// TIA Portal project "E01_KOP_SCL" (V18)

(* hardware
DEVICE "S71500/ET200MP station_1"  S7-1500 station
   slot 0: "Telaio di montaggio_0"  Rack  6ES7 590-1***0-0AA0
   slot 1: "PLC_1"  CPU 1516-3 PN/DP  6ES7 516-3AN01-0AB0  V2.5
      slot 3: "Display CPU_1"  6ES7591-1BA00-0AA0
   slot 2: "DI 32x24VDC HF_1"  DI 32x24VDC HF  6ES7 521-1BL00-0AB0  V2.1
   slot 3: "DQ 32x24VDC/0.5A HF_1"  DQ 32x24VDC/0.5A HF  6ES7 522-1BL01-0AB0  V1.0
   slot 4: "AI 8xU/I/RTD/TC ST_1"  AI 8xU/I/RTD/TC ST  6ES7 531-7KF00-0AB0  V2.1
   slot 5: "AQ 4xU/I ST_1"  AQ 4xU/I ST  6ES7 532-5HD00-0AB0  V2.1
*)

// ===== PLC "PLC_1"  CPU 1516-3 PN/DP =====

VAR_GLOBAL   // PLC tag table "Tabella delle variabili standard"
   "Led 1" AT %Q3.0 : Bool;
   "Led 2" AT %Q3.1 : Bool;
   "Led 3" AT %Q3.2 : Bool;
   "Led 4" AT %Q3.3 : Bool;
   "Led 5" AT %Q3.4 : Bool;
   "Led 6" AT %Q3.5 : Bool;
   "Led 7" AT %Q3.6 : Bool;
   "Led 8" AT %Q3.7 : Bool;
END_VAR

DATA_BLOCK "DB_dati"   // DB1
{ S7_Optimized_Access := 'TRUE' }
VERSION : 0.1
   VAR
      btn1 : Bool;
      btn2 : Bool;
      btn3 : Bool;
      btn4 : Bool;
      btn5 : Bool;
      btn6 : Bool;
      btn7 : Bool;
      btn8 : Bool;
   END_VAR
BEGIN
END_DATA_BLOCK

FUNCTION "FC_KOP" : Void   // FC1, LAD
{ S7_Optimized_Access := 'TRUE' }
VERSION : 0.1
BEGIN

REGION Network 1
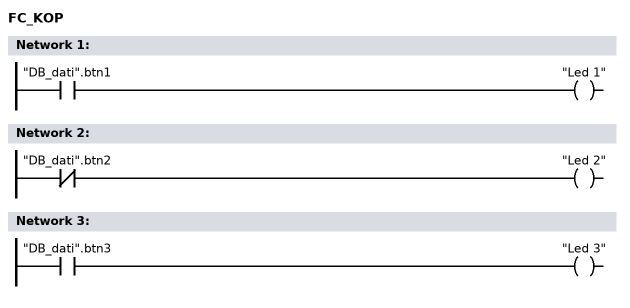
   RUNG wire#powerrail
      Contact( "DB_dati".btn1 )
      Coil( "Led 1" )
   END_RUNG
   // the same network as SCL:
   "Led 1" := "DB_dati".btn1;
END_REGION

REGION Network 2
   RUNG wire#powerrail
      I_Contact( "DB_dati".btn2 )
      Coil( "Led 2" )
   END_RUNG
   // the same network as SCL:
   "Led 2" := NOT "DB_dati".btn2;
END_REGION

REGION Network 3
   RUNG wire#powerrail
      Contact( "DB_dati".btn3 )
      Coil( "Led 3" )
   END_RUNG
   // the same network as SCL:
   "Led 3" := "DB_dati".btn3;
END_REGION
END_FUNCTION

FUNCTION "FC_SCL" : Void   // FC2, SCL
{ S7_Optimized_Access := 'TRUE' }
VERSION : 0.1
BEGIN
   IF "DB_dati".btn4 = TRUE THEN
       "Led 4" := TRUE;
   ELSE
       "Led 4" := FALSE;
   END_IF;
   //Commenti 
   IF "DB_dati".btn5 = FALSE THEN
       "Led 5" := TRUE;
   ELSE
       "Led 5" := FALSE;
   END_IF;
   //
   IF "DB_dati".btn6 = TRUE THEN
       "Led 6" := TRUE;
   ELSE
       "Led 6" := FALSE;
   END_IF;
END_FUNCTION

ORGANIZATION_BLOCK "Main"   // OB1, LAD, ProgramCycle
TITLE = "Main Program Sweep (Cycle)"
{ S7_Optimized_Access := 'TRUE' }
VERSION : 0.1
   VAR_INPUT
      Initial_Call : Bool;   // Initial call of this OB
      Remanence : Bool;   // =True, if remanent data are available
   END_VAR
   VAR_TEMP   // added for the SCL form of the ladder/FBD networks
      _w1 : Bool;
   END_VAR
BEGIN

REGION Network 1
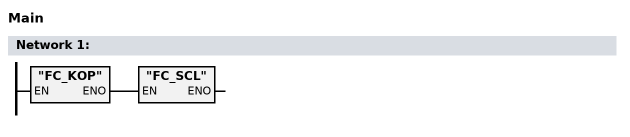
   RUNG wire#powerrail
      "FC_KOP"()
      "FC_SCL"()
   END_RUNG
   // the same network as SCL:
   "FC_KOP"(ENO => #_w1);
   IF #_w1 THEN "FC_SCL"(); END_IF;
END_REGION
END_ORGANIZATION_BLOCK